{attribute 'reflection'}
FUNCTION_BLOCK FB_MatrixSubMatrix_Test EXTENDS FB_TestSuite
VAR_INPUT
END_VAR
VAR_OUTPUT
END_VAR
VAR
END_VAR

WhenCreatedExpectDataRetained();

METHOD PRIVATE WhenCreatedExpectDataRetained
VAR_INPUT
END_VAR
VAR
	M1 : DynamicMatrix;
	M2 : DynamicMatrix;
	Result : BOOL;
	
	Ri : UINT;
	Ci : UINT;
	
	Expected : LREAL;
	Actual : LREAL;
END_VAR
TEST('WhenCreatedExpectDataRetained');

// @TEST-RUN
M1.InitMagicSquare(5);
Result := M2.AsSubMatrix(M1,1,3,1,3);

// @TEST-ASSERT
AssertTrue(Result,'Main function call was not successful');

FOR Ri := 0 TO M2.Rows-1 DO
	FOR Ci := 0 TO M2.Cols-1 DO
		Expected := M1.GetRC(Ri+1,Ci+1);
		Actual := M2.GetRC(Ri,Ci);
		AssertEquals(Expected, Actual, 'Equivalent values are not equal after submatrix');
	END_FOR;
END_FOR

TEST_FINISHED();
END_METHOD

END_FUNCTION_BLOCK

(* stored: Version 1.1.0.1, ProductVersion 3.1.4024.9
   POU FB_MatrixSubMatrix_Test: Id {ef45b795-bcc1-0b30-385f-8eea9a7a6ef8}, SpecialFunc None
   Method WhenCreatedExpectDataRetained: Id {88f20cd2-8fe8-057d-2917-50566d2adf1e} *)
